{attribute 'qualified_only'}
VAR_GLOBAL
	iMainFrame 		: INT;
	bReset			: BOOL;
	bRun			: BOOL;
	bInit			: BOOL;
	bAging_test		: BOOL;
END_VAR

(* stored: Version 1.1.0.1, ProductVersion 3.1.4024.12
   GVL G_HMI: Id {1f28405a-7fc1-4023-8e02-e5a4478b4d4e} *)
